{attribute 'no_explicit_call' := 'do not call this POU directly'} 
FUNCTION_BLOCK SensorBeckhoff IMPLEMENTS ISensor, __SYSTEM.IQueryInterface
VAR
	io_in			: REFERENCE TO SensorBeckhoffIO_in;
	_value			: LREAL;
	
	inputMin		: LREAL;
	inputMax		: LREAL;
	outputMin		: LREAL;
	outputMax		: LREAL;
END_VAR

METHOD FB_init : BOOL
VAR_INPUT
	bInitRetains : BOOL; // if TRUE, the retain variables are initialized (warm start / cold start)
	bInCopyCode : BOOL;  // if TRUE, the instance afterwards gets moved into the copy code (online change)
	IO_in			: REFERENCE TO SensorBeckhoffIO_in;
	InputMin		: LREAL;
	InputMax		: LREAL;
	OutputMin		: LREAL;
	OutputMax		: LREAL;
END_VAR
THIS^.io_in REF= IO_in;
THIS^.inputMin := InputMin;
THIS^.inputMax := InputMax;
THIS^.outputMin := OutputMin;
THIS^.outputMax := OutputMax;
END_METHOD

METHOD update : BOOL
_value := transform(TO_LREAL(io_in.ValuesRaw), inputMin, inputMax, outputMin, outputMax, LimitY := TRUE);
END_METHOD

PROPERTY Value : LREAL
GET
Value := _value;
END_GET
END_PROPERTY

END_FUNCTION_BLOCK

(* stored: Version 1.1.0.1
   POU SensorBeckhoff: Id {8d8bb85b-494f-0dfa-243d-888aa5e878a2}, SpecialFunc None
   Method FB_init: Id {0a9ff2f6-5677-023e-37fd-430c5cf6eb66}
   Method update: Id {476afc7e-048b-02d8-1126-cfcbe86c5a52}
   Property Value: Id {c421dfad-fa40-0144-09ff-143801054b78}
   Get Get: Id {c8851d03-277c-0800-250f-b862d105cbc1} *)
